// TIA Portal V20 export
TYPE "SHIFTMODEL_LIST_UDT"
   STRUCT
      ShiftmodelList_Zero { ExternalAccessible := 'False'; ExternalVisible := 'False'; ExternalWritable := 'False'; S7_SetPoint := 'True'} : "SHIFTMODEL-TIMES_1DAY_UDT";   // Alle Zeitwerte (TOD) gleich 00:00:00 / All Time values (TOD) are 00:00:00
      ShiftmodelList_1 { ExternalAccessible := 'False'; ExternalVisible := 'False'; ExternalWritable := 'False'; S7_SetPoint := 'True'} : "SHIFTMODEL-TIMES_1DAY_UDT";   // Schichtmodel Liste 1 (1 Tag) / Shiftmodel list 1 (1 day)
      ShiftmodelList_2 { ExternalAccessible := 'False'; ExternalVisible := 'False'; ExternalWritable := 'False'; S7_SetPoint := 'True'} : "SHIFTMODEL-TIMES_1DAY_UDT";   // Schichtmodel Liste 2 (1 Tag) / Shiftmodel list 2 (1 day)
      ShiftmodelList_3 { ExternalAccessible := 'False'; ExternalVisible := 'False'; ExternalWritable := 'False'; S7_SetPoint := 'True'} : "SHIFTMODEL-TIMES_1DAY_UDT";   // Schichtmodel Liste 3 (1 Tag) / Shiftmodel list 3 (1 day)
      ShiftmodelList_4 { ExternalAccessible := 'False'; ExternalVisible := 'False'; ExternalWritable := 'False'; S7_SetPoint := 'True'} : "SHIFTMODEL-TIMES_1DAY_UDT";   // Schichtmodel Liste 4 (1 Tag) / Shiftmodel list 4 (1 day)
      ShiftmodelList_5 { ExternalAccessible := 'False'; ExternalVisible := 'False'; ExternalWritable := 'False'; S7_SetPoint := 'True'} : "SHIFTMODEL-TIMES_1DAY_UDT";   // Schichtmodel Liste 5 (1 Tag) / Shiftmodel list 5 (1 day)
      ShiftmodelList_6 { ExternalAccessible := 'False'; ExternalVisible := 'False'; ExternalWritable := 'False'; S7_SetPoint := 'True'} : "SHIFTMODEL-TIMES_1DAY_UDT";   // Schichtmodel Liste 6 (1 Tag) / Shiftmodel list 6 (1 day)
      ShiftmodelList_7 { ExternalAccessible := 'False'; ExternalVisible := 'False'; ExternalWritable := 'False'; S7_SetPoint := 'True'} : "SHIFTMODEL-TIMES_1DAY_UDT";   // Schichtmodel Liste 7 (1 Tag) / Shiftmodel list 7 (1 day)
      ShiftmodelList_8 { ExternalAccessible := 'False'; ExternalVisible := 'False'; ExternalWritable := 'False'; S7_SetPoint := 'True'} : "SHIFTMODEL-TIMES_1DAY_UDT";   // Schichtmodel Liste 8 (1 Tag) / Shiftmodel list 8 (1 day)
      ShiftmodelList_9 { ExternalAccessible := 'False'; ExternalVisible := 'False'; ExternalWritable := 'False'; S7_SetPoint := 'True'} : "SHIFTMODEL-TIMES_1DAY_UDT";   // Schichtmodel Liste 9 (1 Tag) / Shiftmodel list 9 (1 day)
      ShiftmodelList_10 { ExternalAccessible := 'False'; ExternalVisible := 'False'; ExternalWritable := 'False'; S7_SetPoint := 'True'} : "SHIFTMODEL-TIMES_1DAY_UDT";   // Schichtmodel Liste 10 (1 Tag) / Shiftmodel list 10 (1 day)
      Shiftmodel_WeekDay { ExternalAccessible := 'False'; ExternalVisible := 'False'; ExternalWritable := 'False'; S7_SetPoint := 'True'} : Array[1..7] of "SHIFTMODEL-TIMES_1DAY_UDT";   // Schichtmodel 1 Woche (1: Sunday, 2: Monday, 3: Thuesday, 4: Wednesday, 5: Thursday, 6: Friday, 7: Saturday) / Shiftmodel 1 week (1: Sunday, 2: Monday, 3: Thuesday, 4: Wednesday, 5: Thursday, 6: Friday, 7: Saturday)
   END_STRUCT;
END_TYPE
